PROGRAM POU_1
VAR
	
	objectDetected : BOOL := FALSE;

	blackObject : BOOL := FALSE;	
	redObject : BOOL := FALSE;
	
	motorOn : BOOL := FALSE;
	actuatorMove : BOOL := FALSE;
	
	objectSorted : BOOL := FALSE;
	
	startTimer : BOOL := FALSE;
	TON_0: TON;
	
END_VAR

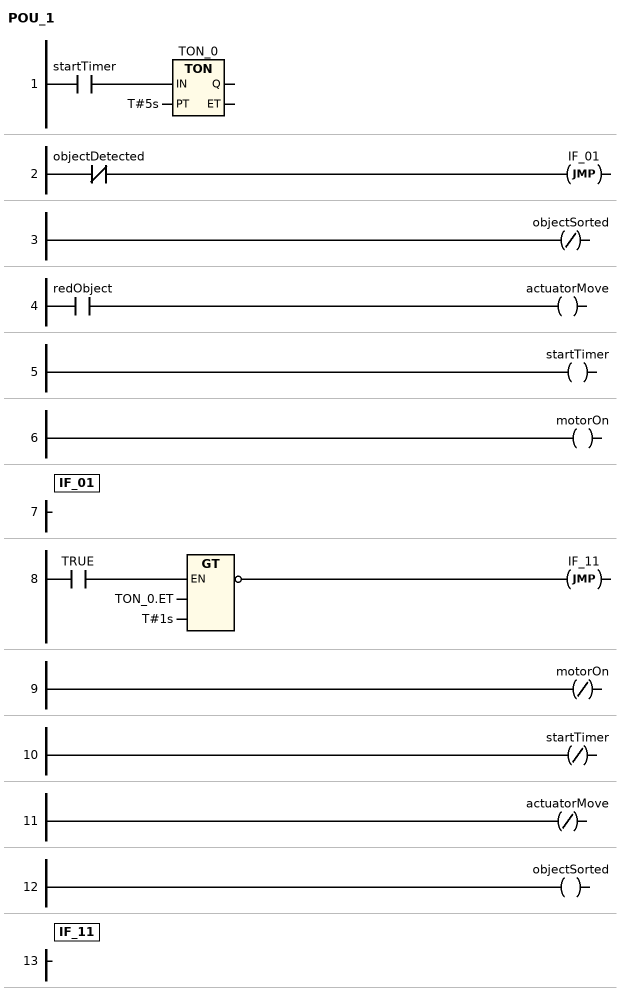
// NETWORK 1
TON_0(IN := startTimer, PT := T#5s); // TON

// NETWORK 2
IF NOT objectDetected THEN JMP IF_01; END_IF

// NETWORK 3
objectSorted := NOT TRUE;

// NETWORK 4
actuatorMove := redObject;

// NETWORK 5
startTimer := TRUE;

// NETWORK 6
motorOn := TRUE;

// NETWORK 7
IF_01: ;

// NETWORK 8
IF NOT (TON_0.ET > T#1s) THEN JMP IF_11; END_IF

// NETWORK 9
motorOn := NOT TRUE;

// NETWORK 10
startTimer := NOT TRUE;

// NETWORK 11
actuatorMove := NOT TRUE;

// NETWORK 12
objectSorted := TRUE;

// NETWORK 13
IF_11: ;

END_PROGRAM

(* stored: Version 1.1.0.1, ProductVersion 3.1.4024.3
   POU POU_1: Id {3648c217-7e4a-40c1-9da7-5ce41d76ddb1}, SpecialFunc None *)
